// TIA Portal V18 export
FUNCTION "LT_GT_OK" : Void   // FC16, FBD
{ S7_Optimized_Access := 'TRUE' }
VERSION : 0.1
// stored: AutoNumber true, IsIECCheckEnabled false, SetENOAutomatically false, UDAEnableTagReadback false
   VAR_INPUT
      value : Real;
      min : Real;
      max : Real;
   END_VAR
   VAR_OUTPUT
      OK : Bool;
      LT_MIN : Bool;
      GT_MAX : Bool;
   END_VAR
BEGIN

REGION Network 1
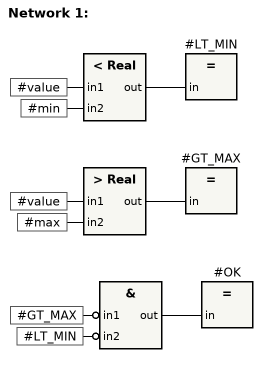
   #LT_MIN := #value < #min;
   #GT_MAX := #value > #max;
   #OK := NOT #GT_MAX AND NOT #LT_MIN;
END_REGION
END_FUNCTION
